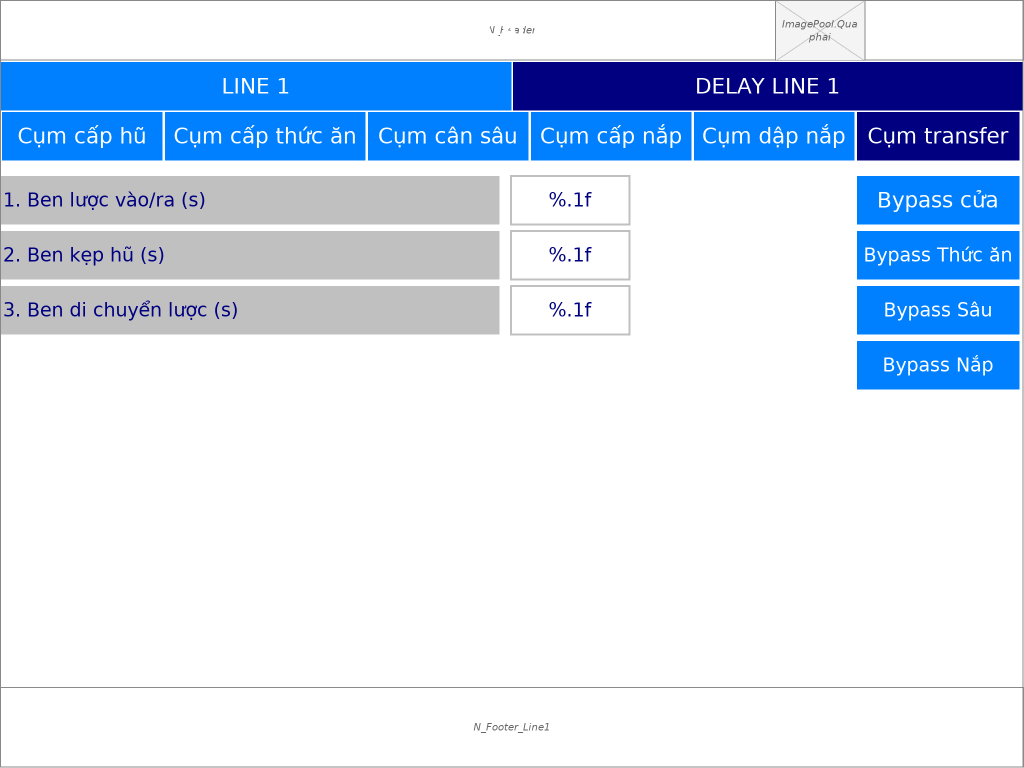
VISUALIZATION N_Setting_Delay_Tranfer1  // 1024x768
    Frame (0,687 1024x80)
        shows N_Footer_Line1()
    Frame (0,0 1024x60)
        shows N_Header()
    Textfield (353,4 420x50), "MÀN HÌNH CÀI KHOẢNG TRỄ LINE 1"
    Rectangle (0,61 512x50), "LINE 1"
        OnMouseClick: change screen: N_Setting_Line1
    Image (775,0 90x61), image: ImagePool.Qua phai
        OnMouseClick: change screen: N_Setting_Delay_Tranfer2
    Rectangle (0,230 500x50), "2. Ben kẹp hũ (s)"
    Rectangle (0,285 500x50), "3. Ben di chuyển lược (s)"
    Rectangle (510,175 120x50), "%.1f", text variable: PR_Line01.fTimer_Comb
        OnMouseClick: write PR_Line01.fTimer_Comb via VisuDialogs.Numpad
    Rectangle (510,230 120x50), "%.1f", text variable: PR_Line01.fTimer_Clip
        OnMouseClick: write PR_Line01.fTimer_Clip via VisuDialogs.Numpad
    Rectangle (510,285 120x50), "%.1f", text variable: PR_Line01.fTimer_Move_Comb
        OnMouseClick: write PR_Line01.fTimer_Move_Comb via VisuDialogs.Numpad
    Rectangle (1,111 162x50), "Cụm cấp hũ"
        OnMouseClick: change screen: N_Setting_Delay_JarSupply1
    Rectangle (164,111 202x50), "Cụm cấp thức ăn"
        OnMouseClick: change screen: N_Setting_Delay_FoodSupply1
    Rectangle (367,111 162x50), "Cụm cân sâu"
        OnMouseClick: change screen: N_Setting_Delay_WormWeight1
    Rectangle (530,111 162x50), "Cụm cấp nắp"
        OnMouseClick: change screen: N_Setting_Delay_LidSupply1
    Rectangle (693,111 162x50), "Cụm dập nắp"
        OnMouseClick: change screen: N_Setting_Delay_LidPressing1
    Rectangle (856,111 164x50), "Cụm transfer"
        OnMouseClick: change screen: N_Setting_Delay_Tranfer1
    Rectangle (512,61 511x50), "DELAY LINE 1"
        OnMouseClick: change screen: N_Setting_Delay_JarSupply1
    Rectangle (0,175 500x50), "1. Ben lược vào/ra (s)"
    Rectangle (856,175 164x50), "Bypass cửa"
        toggle bypass
    Rectangle (856,230 164x50), "Bypass Thức ăn"
        toggle PR_Line01.bypassfood
    Rectangle (856,285 164x50), "Bypass Sâu"
        toggle PR_Line01.bypassWorm
    Rectangle (856,340 164x50), "Bypass Nắp"
        toggle PR_Line01.bypassLid
END_VISUALIZATION

(* stored: Version 1.1.0.1, ProductVersion 3.1.4024.12
   Visu N_Setting_Delay_Tranfer1: Id {a3dd1867-bf46-4d7d-91db-bef383062d81} *)
